Staubli VAL3: onInsert.pgx

public program onInsert(string& x_sItem[])
  local string l_sEvent
begin
  cls()
  // select the type
  call selectType(l_sEvent)
  // exit
  if l_sEvent==""
    return
  else
    // copy it
    x_sItem=l_sEvent
  endIf
  // make it
  call make_it(x_sItem)
  //
end
